// TIA Portal project "Loop_Traffic_Light_V1" (V18)

(* hardware
DEVICE "S7-1500/ET200MP station_1"  S7-1500 station
   slot 0: "导轨_0"  Rack  6ES7 590-1***0-0AA0
   slot 1: "PLC_1"  CPU 1516-3 PN/DP  6ES7 516-3AN01-0AB0  V2.6
      slot 3: "CPU 显示_1"  6ES7591-1BA00-0AA0
      slot 32768: "PROFINET 接口_1"  X1
      slot 33024: "PROFINET 接口_2"  X2
      slot 33280: "DP 接口_1"  X3
   slot 2: "DI 32x24VDC HF_1"  DI 32x24VDC HF  6ES7 521-1BL00-0AB0  V2.1
   slot 3: "DQ 32x24VDC/0.5A HF_1"  DQ 32x24VDC/0.5A HF  6ES7 522-1BL01-0AB0  V1.1
   slot 4: "AI 8xU/I/RTD/TC ST_1"  AI 8xU/I/RTD/TC ST  6ES7 531-7KF00-0AB0  V2.2
   slot 5: "AQ 4xU/I ST_1"  AQ 4xU/I ST  6ES7 532-5HD00-0AB0  V2.2
DEVICE "HMI_1"  TP700 Comfort
   slot 0: "HMI_1"  TP700 Comfort  6AV2 124-0GC01-0AX0  15.1.0.0
   slot 1: "HMI_RT_1"  TP700 Comfort  6AV2 124-0GC01-0AX0  15.1.0.0
   slot 5: "HMI_1.IE_CP_1"  PROFINET Interface  15.0.1.0
      slot 1: "PROFINET Interface_1"  PROFINET Interface
         slot 1: "Port_1"  Port
         slot 2: "Port_2"  Port
   slot 7: "HMI_1.MPI/DP_CP_1"  MPI/DP Interface  15.0.1.0
*)

// ===== PLC "PLC_1"  CPU 1516-3 PN/DP =====

VAR_GLOBAL   // PLC tag table "默认变量表"
   "System_Byte" AT %MB1 : Byte;
   "FirstScan" AT %M1.0 : Bool;
   "DiagStatusUpdate" AT %M1.1 : Bool;
   "AlwaysTRUE" AT %M1.2 : Bool;
   "AlwaysFALSE" AT %M1.3 : Bool;
   "Clock_Byte" AT %MB0 : Byte;
   "Clock_10Hz" AT %M0.0 : Bool;
   "Clock_5Hz" AT %M0.1 : Bool;
   "Clock_2.5Hz" AT %M0.2 : Bool;
   "Clock_2Hz" AT %M0.3 : Bool;
   "Clock_1.25Hz" AT %M0.4 : Bool;
   "Clock_1Hz" AT %M0.5 : Bool;
   "Clock_0.625Hz" AT %M0.6 : Bool;
   "Clock_0.5Hz" AT %M0.7 : Bool;
   "红灯亮10s" AT %M2.0 : Bool;
   "黄灯亮3s" AT %M2.1 : Bool;
   "绿灯闪烁4s" AT %M2.2 : Bool;
   "按钮A" AT %I1.0 : Bool;
   "按钮B" AT %I1.1 : Bool;
END_VAR

DATA_BLOCK "工序"   // DB1
{ S7_Optimized_Access := 'TRUE' }
VERSION : 0.1
   VAR
      执行序数 : Int;
      循环次数 : Int;
      灯状态 : Int;
   END_VAR
BEGIN
END_DATA_BLOCK

// folder: System blocks/Program resources

DATA_BLOCK "T1"   // DB2
{ S7_Optimized_Access := 'TRUE' }
AUTHOR : Simatic
FAMILY : IEC
NAME : IEC_TMR
VERSION : 1.0
// stored: InstanceOfName IEC_TIMER
"IEC_TIMER"
BEGIN
END_DATA_BLOCK

DATA_BLOCK "T2"   // DB3
{ S7_Optimized_Access := 'TRUE' }
AUTHOR : Simatic
FAMILY : IEC
NAME : IEC_TMR
VERSION : 1.0
// stored: InstanceOfName IEC_TIMER
"IEC_TIMER"
BEGIN
END_DATA_BLOCK

DATA_BLOCK "T3"   // DB4
{ S7_Optimized_Access := 'TRUE' }
AUTHOR : Simatic
FAMILY : IEC
NAME : IEC_TMR
VERSION : 1.0
// stored: InstanceOfName IEC_TIMER
"IEC_TIMER"
BEGIN
END_DATA_BLOCK

// folder: (top level)

ORGANIZATION_BLOCK "Main"   // OB1, LAD, ProgramCycle
TITLE = "Main Program Sweep (Cycle)"
{ S7_Optimized_Access := 'TRUE' }
VERSION : 0.1
   VAR_INPUT
      Initial_Call : Bool;   // Initial call of this OB
      Remanence : Bool;   // =True, if remanent data are available
   END_VAR
BEGIN

REGION Network 1
   // 上课跟着敲的
   // 1.避免双线圈
   // 2.写顺序结构--->工序进行程序隔离
   // 3.顺序的基本架构和执行分开来写
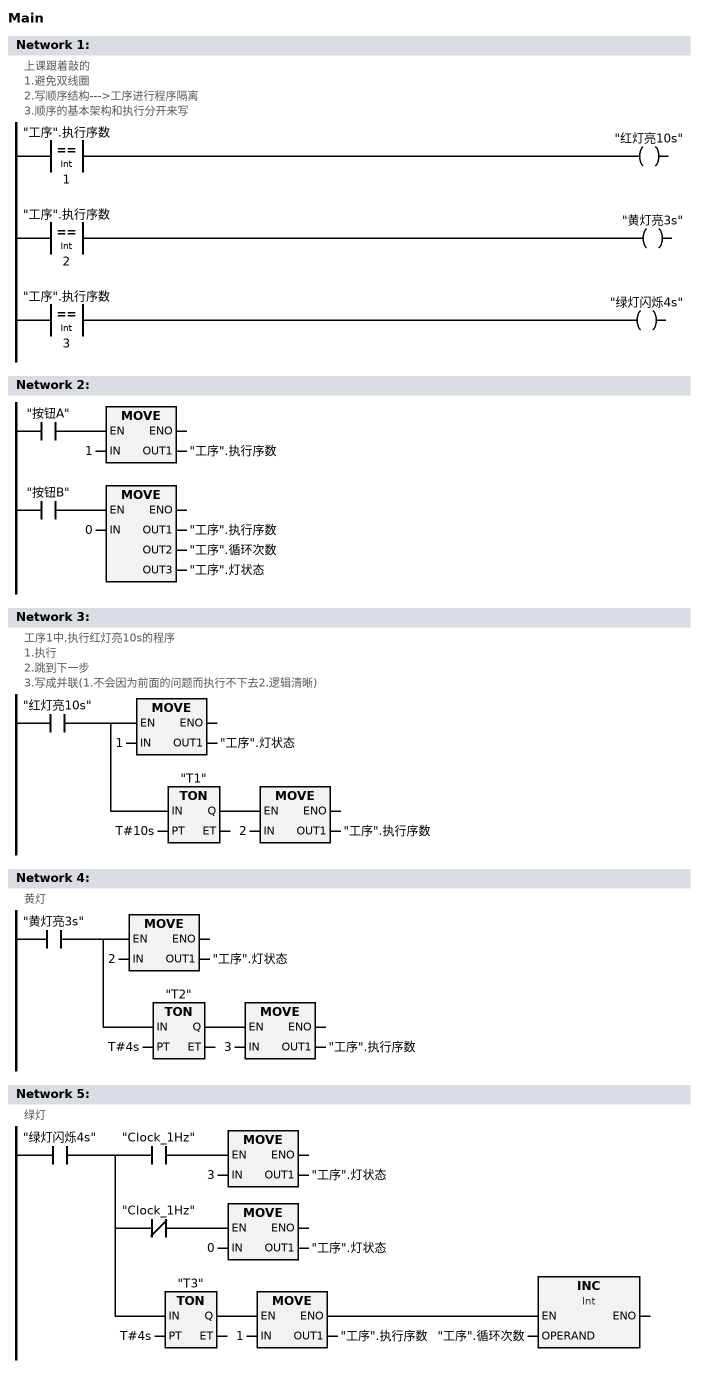
   RUNG wire#powerrail
      { S7_Templates := "SrcType := Int" } EQ_Contact(in1 := "工序".执行序数, in2 := 1)
      Coil( "红灯亮10s" )
   END_RUNG
   RUNG wire#powerrail
      { S7_Templates := "SrcType := Int" } EQ_Contact(in1 := "工序".执行序数, in2 := 2)
      Coil( "黄灯亮3s" )
   END_RUNG
   RUNG wire#powerrail
      { S7_Templates := "SrcType := Int" } EQ_Contact(in1 := "工序".执行序数, in2 := 3)
      Coil( "绿灯闪烁4s" )
   END_RUNG
   // the same network as SCL:
   "红灯亮10s" := "工序".执行序数 = 1;
   "黄灯亮3s" := "工序".执行序数 = 2;
   "绿灯闪烁4s" := "工序".执行序数 = 3;
END_REGION

REGION Network 2
   RUNG wire#powerrail
      Contact( "按钮A" )
      Move(in := 1, out1 => "工序".执行序数)
   END_RUNG
   RUNG wire#powerrail
      Contact( "按钮B" )
      Move(in := 0, out1 => "工序".执行序数, out2 => "工序".循环次数, out3 => "工序".灯状态)
   END_RUNG
   // the same network as SCL:
   IF "按钮A" THEN "工序".执行序数 := 1; END_IF;
   IF "按钮B" THEN
       "工序".执行序数 := 0;
       "工序".循环次数 := 0;
       "工序".灯状态 := 0;
   END_IF;
END_REGION

REGION Network 3
   // 工序1中,执行红灯亮10s的程序
   // 1.执行
   // 2.跳到下一步
   // 3.写成并联(1.不会因为前面的问题而执行不下去2.逻辑清晰)
   IF "红灯亮10s" THEN "工序".灯状态 := 1; END_IF;
   "T1".TON(IN := "红灯亮10s", PT := T#10s);
   IF "T1".Q THEN "工序".执行序数 := 2; END_IF;
END_REGION

REGION Network 4
   // 黄灯
   IF "黄灯亮3s" THEN "工序".灯状态 := 2; END_IF;
   "T2".TON(IN := "黄灯亮3s", PT := T#4s);
   IF "T2".Q THEN "工序".执行序数 := 3; END_IF;
END_REGION

REGION Network 5
   // 绿灯
   IF "绿灯闪烁4s" AND "Clock_1Hz" THEN "工序".灯状态 := 3; END_IF;
   IF "绿灯闪烁4s" AND NOT "Clock_1Hz" THEN "工序".灯状态 := 0; END_IF;
   "T3".TON(IN := "绿灯闪烁4s", PT := T#4s);
   IF "T3".Q THEN
       "工序".执行序数 := 1;
       "工序".循环次数 := "工序".循环次数 + 1;
   END_IF;
END_REGION
END_ORGANIZATION_BLOCK

(* ===== HMI "HMI_RT_1" =====
system functions are stored by id; their names below are inferred from use
connection "HMI_连接_1": ETHERNET, S7_1500_OMS

HMI tags "默认变量表"
   "Tag_ScreenNumber" : UInt, internal
   "按钮A" : Bool = PLC 按钮A AT %I1.0, 100 ms
   "按钮B" : Bool = PLC 按钮B AT %I1.1, 100 ms
   "工序_循环次数" : Int = PLC 工序.循环次数 AT %DB1.DBX0.0, 100 ms
   "工序_灯状态" : Int = PLC 工序.灯状态 AT %DB1.DBX0.0, 100 ms

screen "根画面" 800x420, template "模板_1"
   on GenerateScreen: SetTag("Tag_ScreenNumber", 1)
   Button "按钮_1" at 133,71 size 156x67; TextOff '按钮A'
      on Press: SetBit("按钮A")
      on Release: ResetBit("按钮A")
   Button "按钮_2" at 133,143 size 156x75; TextOff '按钮B'
      on Release: ResetBit("按钮B")
      on Press: SetBit("按钮B")
   Circle "圆_1" at 458,43 size 90x90
      Appearance <- "工序_灯状态"
   IOField "I/O 域_1" at 441,169 size 115x43; FormatPattern 99999
      ProcessValue <- "工序_循环次数"
   TextField "文本域_4" at 576,185 size 73x20; Text '循环次数'

Template "模板_1" 800x420
   Button "退出" at 720,360 size 78x58; TextOff '退出'; PictureOff "ExitRuntime_TP700_Comfort_TR"; PictureOn "ExitRuntime_TP700_Comfort_TR"
      on Release: StopRuntime(0)
   Button "Template_Button" at 640,360 size 78x58; TextOff 'Text'
   Button "Template_Button_1" at 560,360 size 78x58; TextOff 'Text'
   Button "Template_Button_2" at 480,360 size 78x58; TextOff 'Text'
   Button "Template_Button_3" at 400,360 size 78x58; TextOff 'Text'
   Button "Template_Button_4" at 321,360 size 78x58; TextOff 'Text'
   Button "Template_Button_5" at 241,360 size 78x58; TextOff 'Text'
   Button "Template_Button_6" at 161,360 size 78x58; TextOff 'Text'
   Button "报警" at 81,360 size 78x58; TextOff '报警'; PictureOff "AlarmDisplay_TP700_Comfort_TR"; PictureOn "AlarmDisplay_TP700_Comfort_TR"
      on Release: function_ef3f5d25("报警窗口_Unacknowledged", -1)
   Button "起始画面" at 1,360 size 78x58; TextOff '起始画面'; PictureOff "NavigateHome_TP700_Comfort_TR"; PictureOn "NavigateHome_TP700_Comfort_TR"
      on Release: ActivateScreen("根画面", 0)
*)